FUNCTION F_Turbo_NC_NO_Valve_Logic : BOOL
VAR_INPUT
	i_stTurbo : ST_PTM; // Turbo Pump
	i_stISG : ST_VG; //Gauge measuring inlet Pressure e.g Pirani
	i_stBSG : ST_VG; //Gauge measureing backing pressure
	iq_stValve_NO : ST_VRC_NO; //Normally Open Valve directly sharing turbo pump vaccum volume.
	iq_stValve_NC : ST_VRC_NO; //Normally Closed Valve directly sharing turbo pump vaccum volume.
	iq_stValve_NC_second :	ST_VRC_NO; //Normally Closed Valve on the other side of NO valve that also connects to roughing line.
	EcatBridge_Error_Present	:	BOOL; // ADS Communication: Watchdog and ADS Read Error Bit 
	iq_stRoughRoughValve_NC_xOpnLS: BOOL; //Normally Closed Valve Downstream of iq_stValve_NC in Beamline Roughing Line, Open Limit Switch.
	iq_stRoughRoughValve_NC_second_xOpenLS: BOOL; //Normally Closed Valve Downstream of iq_stValve_NC_second in Beamline Roughing Line, Open Limit Switch.
	x_onBeamline :	BOOL; //Whether the  Turbopump/Endstation is mounted on the beamline or not.
END_VAR
VAR
END_VAR

IF (x_onBeamline) THEN
	F_Turbo_NC_NO_Valve_Logic := (i_stISG.xPRESS_OK AND i_stISG.rPRESS < i_stTurbo.rInletPressureSP) AND 
						   		 (i_stBSG.xPRESS_OK AND i_stBSG.rPRESS < i_stTurbo.rBackingPressureSP) AND 
								 ((iq_stValve_NC.i_xOpnLS AND iq_stRoughRoughValve_NC_xOpnLS) OR
								 (iq_stValve_NO.i_xOpnLS AND (iq_stValve_NC_second.i_xOpnLS AND 
								 iq_stRoughRoughValve_NC_second_xOpenLS)))AND (NOT EcatBridge_Error_Present);
ELSE
	F_Turbo_NC_NO_Valve_Logic := (i_stISG.xPRESS_OK AND i_stISG.rPRESS < i_stTurbo.rInletPressureSP) AND 
						   (i_stBSG.xPRESS_OK AND i_stBSG.rPRESS < i_stTurbo.rBackingPressureSP) AND 
							(iq_stValve_NC.i_xOpnLS OR(iq_stValve_NO.i_xOpnLS AND iq_stValve_NC_second.i_xOpnLS));
END_IF

END_FUNCTION

(* stored: Version 1.1.0.1, ProductVersion 3.1.4024.6
   POU F_Turbo_NC_NO_Valve_Logic: Id {d3d12688-6a72-46ad-96e0-b6196dc124c6}, SpecialFunc None *)
